FUNCTION TryConvert_TIME_TO_DWORD : BOOL
VAR_INPUT
	in : TIME;
	out : REFERENCE TO DWORD;
END_VAR

out := TIME_TO_DWORD(in);
TryConvert_TIME_TO_DWORD := TRUE;

END_FUNCTION

(* stored: Version 1.1.0.1, ProductVersion 3.1.4024.12
   POU TryConvert_TIME_TO_DWORD: Id {24749b45-7faf-4645-ba03-f7f2b2247cab}, SpecialFunc None *)
